(*
SPDX-FileCopyrightText: © 2026 Oleksandr Tiutyk <trofimich@gmail.com>
SPDX-License-Identifier: MIT
License: https://opensource.org/license/mit
*)

(*!
<summary>Defines an automation component's lifecycle, diagnostics and event delivery capabilities.</summary>
<description>
Every component can receive both bubbling and broadcast events, including roots and leaves. Delivery and
forwarding do not depend on Enabled or operational state; each recipient decides whether to react in its
current state. Being disabled or stopped does not itself stop propagation. Terminal nodes receive an event
without forwarding it; delivery uses the synchronous borrowed IEventDispatcher contract.
</description>
*)

INTERFACE IAutomationComponent EXTENDS
	TOF_Core.INamed,
	TOF_Core.IErrorProvider,
	TOF_Core.IExecutable,
	TOF_Core.IEventDispatcher

(*!
<summary>Disables cyclic execution and invokes disable hooks.</summary>
<description>
Branches also disable their children. Exceptions from disable hooks propagate to the caller without rolling
back prior effects.
</description>
*)
METHOD FINAL Disable
END_METHOD

(*!
<summary>Enables cyclic execution and invokes enable hooks.</summary>
<description>
Enabling does not automatically reset a STOPPED component. Components stopped while disabled or disabled
while stopped remain STOPPED after Enable until explicitly Reset. Child enablement also enables disabled
parents with includeChildren := FALSE.
</description>
<param name="includeChildren">When TRUE on a branch, recursively enables child components.</param>
*)
METHOD FINAL Enable
VAR_INPUT
	includeChildren : BOOL := TRUE;
END_VAR
END_METHOD

{attribute 'monitoring' := 'call'}
PROPERTY Enabled : BOOL
GET
END_GET
END_PROPERTY

METHOD FINAL GetEffectiveExceptionHandlingPolicy : TOF_Core.IExceptionHandlingPolicy
END_METHOD

(*!
<summary>Sets the maximum wait for pending initialization.</summary>
<description>
T#0S selects Parameters.InitializationTimeout immediately upon assignment, so the getter always returns the
active non-zero duration. During initialization, a branch expands its effective initialization timeout to at
least the maximum InitializationTimeout of its children.
</description>
*)
{attribute 'monitoring' := 'call'}
PROPERTY InitializationTimeout : TIME
GET
END_GET
SET
END_SET
END_PROPERTY

(*!
<summary>Advances initialization after validating mandatory dependencies.</summary>
<description>
Child components require a live constructor-bound parent. Missing required dependencies fail before
initialization hooks. FALSE reports pending work or failure; INVALID never reports TRUE. Caught failures
record a copied critical error in terminal INVALID. Already initialized or stopped components report TRUE.
Completed callback effects are not rolled back.
Only a pending call evaluates the timeout. Completion on the deadline cycle succeeds.
</description>
*)
METHOD Initialize : BOOL
END_METHOD

{attribute 'monitoring' := 'call'}
PROPERTY FINAL OperationalState : OPERATIONAL_STATE
GET
END_GET
END_PROPERTY

{attribute 'monitoring' := 'call'}
PROPERTY FINAL OperationalStateReason : REFERENCE TO WSTRING(255)
GET
END_GET
END_PROPERTY

(*!
<summary>Attempts to recover an enabled stopped component to WORKING.</summary>
<description>
Served only while Enabled and in OPERATIONAL_STATE.STOPPED. Clears the execution error before reset hooks.
A failure in the component's own reset hook (OnReset, OnBeforeChildrenReset or OnAfterChildrenReset) always
leaves the component in OPERATIONAL_STATE.STOPPED with a copied CRITICAL error without consulting the
exception handling policy.
</description>
*)
METHOD Reset
END_METHOD

(*!
<summary>Transitions a WORKING component to OPERATIONAL_STATE.STOPPED.</summary>
<description>
Transitions a WORKING component (and, for branches, all WORKING children) to OPERATIONAL_STATE.STOPPED
regardless of Enabled.
</description>
<param name="reason">Descriptive reason stored in OperationalStateReason.</param>
*)
METHOD FINAL Stop
VAR_INPUT
	reason : WSTRING(255) := "External stop";
END_VAR
END_METHOD

END_INTERFACE

(* stored: Version 1.1.0.1
   Itf IAutomationComponent: Id {b9578ac3-a85d-44ce-81e8-cd1e222e2c39}
   Method Disable: Id {e2aba665-2a02-4877-b9df-ee71836fdfe8}
   Method Enable: Id {ccd0eda5-25b6-4625-9716-04dd6ba8bcd7}
   Property Enabled: Id {01e3c499-4bf3-48d3-b6ca-97f1f477a1ec}
   Get Get: Id {d852fb38-146e-43e8-99a9-7d09aac4a619}
   Method GetEffectiveExceptionHandlingPolicy: Id {b188411a-9a85-4b57-84ff-885a3b56d901}
   Property InitializationTimeout: Id {d3b8e208-f15a-44e7-963c-bb0c332f0ecc}
   Get Get: Id {ba9327c0-e1f7-43df-a35f-6b1ae24b9d23}
   Set Set: Id {226b876b-661d-4572-b4d6-60fb61f56ef1}
   Method Initialize: Id {813191cd-12d8-442d-b7aa-bb11fe623a02}
   Property OperationalState: Id {fcb19fff-e3a4-4b71-a336-7a39fe3f3dd0}
   Get Get: Id {998dd560-089c-49ab-9a99-0cd243d99d71}
   Property OperationalStateReason: Id {75dd6472-8320-43b0-aa1a-34d2106e1dc2}
   Get Get: Id {20d87ad5-052f-492f-b00d-842ab8c1646f}
   Method Reset: Id {05122c55-71c6-426f-9d4d-f6c7fcde37fb}
   Method Stop: Id {14f9c654-9d13-4a3d-976b-1ad5d1b543c4} *)
